// TwinCAT 3 PLC project XYStage
// ProgramVersion: 3.1.4023.0
// libraries:
//   Tc2_MC2, * (Beckhoff Automation GmbH)
//   Tc2_MC2_Drive, * (Beckhoff Automation GmbH)
//   Tc2_Standard, * (Beckhoff Automation GmbH)
//   Tc2_System, * (Beckhoff Automation GmbH)
//   Tc3_Module, * (Beckhoff Automation GmbH)
// project tree:
//   GVLs/ GVL.TcGVL (not stored)
//   / PlcTask.TcTTO (not stored)
//   POUs/ Get_PID_Gain.TcPOU (not stored), MAIN.TcPOU, Init_Devices.TcPOU (not stored)
// real-time tasks:
//   TASK PlcTask: cycle T#10ms, priority 20, ADS port 350
// motion (NC):
//   TASK NC-Task 1 SAF: cycle T#2ms, priority 4, ADS port 501
//   TASK NC-Task 1 SVB: cycle T#10ms, priority 8, ADS port 511
//   AXIS XAxis (id 1)
//     PositionAreaControl: Enable=false
//     OtherSettings: AllowMotionCmdToSlave=true
//     encoder EncType=19
//       EncPara: ScaleFactorNumerator=0.0006, MaxCount=#xffffffff
//     drive DrvType=16
//       DrvPara: MaxCount=#xffffffff, DriveControlDWord=#x00020100
//         Analog: TorqueSetpointScale=10, ScaleFactorActTorque=0.1
//         TimeComp: TaskDelayCycles=1
//     controller CtrType=1
//       CtrPara: PriorControlFactor=1
//         PosDiffControl: Enable=false
//         Observer: BandWidth=20
//   AXIS YAxis (id 2)
//     PositionAreaControl: Enable=false
//     OtherSettings: AllowMotionCmdToSlave=true
//     encoder EncType=19
//       EncPara: ScaleFactorNumerator=0.0006, MaxCount=#xffffffff
//     drive DrvType=16
//       DrvPara: MaxCount=#xffffffff, DriveControlDWord=#x00020100
//         Analog: TorqueSetpointScale=10, ScaleFactorActTorque=0.1
//         TimeComp: TaskDelayCycles=1
//     controller CtrType=1
//       CtrPara: PriorControlFactor=1
//         PosDiffControl: Enable=false
//         Observer: BandWidth=20
// I/O:
//   DEVICE Device 1 (EtherCAT), AmsNetId 5.33.182.40.2.1
//     Term 1 (EK1200) [EK1200-5000 EtherCAT Power supply (2A E-Bus)]
//       Term 2 (EL1018) [EL1018 8Ch. Dig. Input 24V, 10µs]
//       Term 3 (EL2024) [EL2024 4Ch. Dig. Output 24V, 2A]
//       Term 4 (EK1110) [EK1110 EtherCAT extension]
//     Drive 5 (MADLN05BE) [MADLN05BE]
//     Drive 6 (MADLN05BE) [MADLN05BE]
// variable links:
//   NC-Task 1 SAF/Axes/XAxis <-> Device 1 (EtherCAT)/Drive 5 (MADLN05BE)
//     Drive/Inputs/In/nDataIn1 <-> Transmit PDO mapping 1/Following error actual value
//     Drive/Inputs/In/nState1 <-> Transmit PDO mapping 1/Statusword
//     Drive/Inputs/In/nState2 <-> Transmit PDO mapping 1/Statusword @bit 8
//     Drive/Inputs/In/nState4 @bit 1 <-> WcState/InputToggle
//     Drive/Inputs/In/nState4 <-> WcState/WcState
//     Drive/Inputs/In/nState5 <-> Transmit PDO mapping 1/Modes of operation display
//     Drive/Outputs/Out/nCtrl1 <-> Receive PDO mapping 1/Controlword
//     Drive/Outputs/Out/nCtrl2 <-> Receive PDO mapping 1/Controlword @bit 8
//     Drive/Outputs/Out/nCtrl5 <-> Receive PDO mapping 1/Modes of operation
//     Drive/Outputs/Out/nDataOut1 <-> Receive PDO mapping 1/Target position
//     Enc/Inputs/In/nDataIn1 <-> Transmit PDO mapping 1/Position actual value
//     Enc/Inputs/In/nDataIn3 <-> Transmit PDO mapping 1/Touch probe pos1 pos value
//     Enc/Inputs/In/nState4 @bit 1 <-> WcState/InputToggle
//     Enc/Inputs/In/nState4 <-> WcState/WcState
//     Enc/Inputs/In/nState5 <-> Transmit PDO mapping 1/Touch probe status
//     Enc/Inputs/In/nState6 <-> Transmit PDO mapping 1/Touch probe status @bit 8
//     Enc/Outputs/Out/nCtrl5 <-> Receive PDO mapping 1/Touch probe function
//     Enc/Outputs/Out/nCtrl6 <-> Receive PDO mapping 1/Touch probe function @bit 8
//   NC-Task 1 SAF/Axes/YAxis <-> Device 1 (EtherCAT)/Drive 6 (MADLN05BE)
//     Drive/Inputs/In/nDataIn1 <-> Transmit PDO mapping 1/Following error actual value
//     Drive/Inputs/In/nState1 <-> Transmit PDO mapping 1/Statusword
//     Drive/Inputs/In/nState2 <-> Transmit PDO mapping 1/Statusword @bit 8
//     Drive/Inputs/In/nState4 @bit 1 <-> WcState/InputToggle
//     Drive/Inputs/In/nState4 <-> WcState/WcState
//     Drive/Inputs/In/nState5 <-> Transmit PDO mapping 1/Modes of operation display
//     Drive/Outputs/Out/nCtrl1 <-> Receive PDO mapping 1/Controlword
//     Drive/Outputs/Out/nCtrl2 <-> Receive PDO mapping 1/Controlword @bit 8
//     Drive/Outputs/Out/nCtrl5 <-> Receive PDO mapping 1/Modes of operation
//     Drive/Outputs/Out/nDataOut1 <-> Receive PDO mapping 1/Target position
//     Enc/Inputs/In/nDataIn1 <-> Transmit PDO mapping 1/Position actual value
//     Enc/Inputs/In/nDataIn3 <-> Transmit PDO mapping 1/Touch probe pos1 pos value
//     Enc/Inputs/In/nState4 @bit 1 <-> WcState/InputToggle
//     Enc/Inputs/In/nState4 <-> WcState/WcState
//     Enc/Inputs/In/nState5 <-> Transmit PDO mapping 1/Touch probe status
//     Enc/Inputs/In/nState6 <-> Transmit PDO mapping 1/Touch probe status @bit 8
//     Enc/Outputs/Out/nCtrl5 <-> Receive PDO mapping 1/Touch probe function
//     Enc/Outputs/Out/nCtrl6 <-> Receive PDO mapping 1/Touch probe function @bit 8
//   XYStage/XYStage Instance <-> NC-Task 1 SAF/Axes/XAxis
//     PlcTask Inputs/GVL.AxisX.NcToPlc <-> Outputs/ToPlc
//     PlcTask Outputs/GVL.AxisX.PlcToNc <-> Inputs/FromPlc
//   XYStage/XYStage Instance <-> NC-Task 1 SAF/Axes/YAxis
//     PlcTask Inputs/GVL.AxisY.NcToPlc <-> Outputs/ToPlc
//     PlcTask Outputs/GVL.AxisY.PlcToNc <-> Inputs/FromPlc

// ---- POUs/MAIN.TcPOU
PROGRAM MAIN
VAR
		
		
		

END_VAR

// Init
Init_Devices();
//
Get_PID_Gain();


GVL.AxisX_Power_Fuc.Enable := GVL.OnMoterX;
GVL.AxisY_Power_Fuc.Enable := GVL.OnMoterY;



GVL.AxisX_AbMove_Fuc.Execute := GVL.X_AbMove_Ex;
GVL.X_AbMove_Ex := FALSE;


GVL.AxisY_AbMove_Fuc.Execute := GVL.Y_AbMove_Ex;
GVL.Y_AbMove_Ex := FALSE;


GVL.fbCoEWrite_X(
		Axis :=GVL.AxisX,		
		NetId := '5.33.182.40.1.1', 
  		Index := GVL.Index,
  		pSrcBuf := ADR(GVL.X_Gain), 
  		BufLen := SIZEOF(GVL.X_Gain), 
  		Execute := GVL.X_COE_Ex, 
  		Timeout := T#1S, 	
		CompleteAccess := GVL.CompleteAccess, 
		Busy => GVL.Success
	);	
	
GVL.fbCoEWrite_Y(
		Axis :=GVL.AxisY,		
		NetId := '5.33.182.40.1.1', 
  		Index := GVL.Index,
  		pSrcBuf := ADR(GVL.Y_Gain), 
  		BufLen := SIZEOF(GVL.Y_Gain), 
  		Execute := GVL.Y_COE_Ex, 
  		Timeout := T#1S, 	
		CompleteAccess := GVL.CompleteAccess, 
		Busy => GVL.Success
	);

END_PROGRAM
